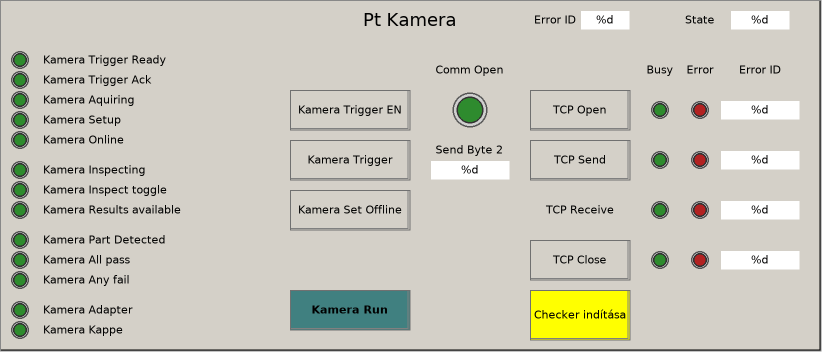
VISUALIZATION Kamera_Pt  // 822x352
    Rectangle (0,0 820x350)
    Lamp1 (450,90 40x40), variable: KAMERAREMOTE.bKameraCommOpen, style: Lamp-Lamp1-Green
    Label (530,200 100x20), "TCP Receive"
    Lamp1 (650,100 20x20), variable: KAMERAREMOTE.bConnectBusy, style: Lamp-Lamp1-Green
    Label (350,0 120x40), "Pt Kamera"
    Button (530,90 100x40), "TCP Open"
        tap KAMERAREMOTE.bKameraCommOpenEnable p1329445385=TRUE
    Button (530,240 100x40), "TCP Close"
        tap KAMERAREMOTE.bKameraCommCloseEnable
    Button (530,140 100x40), "TCP Send"
        tap KAMERAREMOTE.bKameraCommandSend
    Lamp1 (690,100 20x20), variable: KAMERAREMOTE.bConnectError, style: Lamp-Lamp1-Red
    Label (640,60 40x20), "Busy"
    Label (680,60 40x20), "Error"
    Textfield (720,100 80x20), "%d", text variable: KAMERAREMOTE.nConnectErrId
    Label (730,60 60x20), "Error ID"
    Lamp1 (650,250 20x20), variable: KAMERAREMOTE.bCloseBusy, style: Lamp-Lamp1-Green
    Lamp1 (690,250 20x20), variable: KAMERAREMOTE.bCloseError, style: Lamp-Lamp1-Red
    Textfield (720,250 80x20), "%d", text variable: KAMERAREMOTE.nCloseErrId
    Lamp1 (650,150 20x20), variable: KAMERAREMOTE.bSendBusy, style: Lamp-Lamp1-Green
    Lamp1 (690,150 20x20), variable: KAMERAREMOTE.bSendError, style: Lamp-Lamp1-Red
    Textfield (720,150 80x20), "%d", text variable: KAMERAREMOTE.nSendErrId
    Lamp1 (650,200 20x20), variable: KAMERAREMOTE.bReceiveBusy, style: Lamp-Lamp1-Green
    Lamp1 (690,200 20x20), variable: KAMERAREMOTE.bReceiveError, style: Lamp-Lamp1-Red
    Textfield (720,200 80x20), "%d", text variable: KAMERAREMOTE.nReceiveErrId
    Label (430,60 79x20), "Comm Open"
    Label (680,10 40x20), "State"
    Textfield (730,10 60x20), "%d", text variable: KAMERAREMOTE.iState
    Button (290,90 120x40), "Kamera Trigger EN"
        toggle KAMERAREMOTE.bKameraTriggerEN
    Button (290,140 120x40), "Kamera Trigger"
        toggle AUTOMATA.bKameraTrig
    Button (290,190 120x40), "Kamera Set Offline"
        toggle KAMERAREMOTE.bKameraSetOffline
    Textfield (430,160 80x20), "%d", text variable: KAMERAREMOTE.baSendByteArray[2]
    Label (430,140 79x20), "Send Byte 2"
    Label (530,10 50x20), "Error ID"
    Textfield (580,10 50x20), "%d", text variable: KameraProcess.n_OutErrId
    Lamp1 (10,50 20x20), variable: KAMERAREMOTE.bKameraTriggerReady, style: Lamp-Lamp1-Green
    Label (40,50 210x20), "Kamera Trigger Ready"
    Lamp1 (10,70 20x20), variable: KAMERAREMOTE.bKameraTriggerAck, style: Lamp-Lamp1-Green
    Label (40,70 210x20), "Kamera Trigger Ack"
    Lamp1 (10,90 20x20), variable: KAMERAREMOTE.bKameraAcquiring, style: Lamp-Lamp1-Green
    Label (40,90 210x20), "Kamera Aquiring"
    Lamp1 (10,110 20x20), variable: KAMERAREMOTE.bKameraSetup, style: Lamp-Lamp1-Green
    Label (40,110 210x20), "Kamera Setup"
    Lamp1 (10,130 20x20), variable: KAMERAREMOTE.bKameraOnline, style: Lamp-Lamp1-Green
    Label (40,130 210x20), "Kamera Online"
    Lamp1 (10,160 20x20), variable: KAMERAREMOTE.bKameraInspecting, style: Lamp-Lamp1-Green
    Label (40,160 210x20), "Kamera Inspecting"
    Lamp1 (10,180 20x20), variable: KAMERAREMOTE.bKameraInspectToggle, style: Lamp-Lamp1-Green
    Label (40,180 210x20), "Kamera Inspect toggle"
    Lamp1 (10,200 20x20), variable: KAMERAREMOTE.bKameraResultsAvble, style: Lamp-Lamp1-Green
    Label (40,200 210x20), "Kamera Results available"
    Lamp1 (10,230 20x20), variable: KAMERAREMOTE.bKameraPartDetect, style: Lamp-Lamp1-Green
    Label (40,230 210x20), "Kamera Part Detected"
    Lamp1 (10,250 20x20), variable: KAMERAREMOTE.bKameraAllPass, style: Lamp-Lamp1-Green
    Label (40,250 210x20), "Kamera All pass"
    Lamp1 (10,270 20x20), variable: KAMERAREMOTE.bKameraAnyFail, style: Lamp-Lamp1-Green
    Label (40,270 210x20), "Kamera Any fail"
    Lamp1 (10,300 20x20), variable: KAMERAREMOTE.bKameraOut04, style: Lamp-Lamp1-Green
    Label (40,300 210x20), "Kamera Adapter"
    Lamp1 (10,320 20x20), variable: KAMERAREMOTE.bKameraOut05, style: Lamp-Lamp1-Green
    Label (40,320 210x20), "Kamera Kappe"
    Button (290,290 120x40), "Kamera Run"
        toggle KameraProcess.bKameraRun
    Button (530,290 100x50), "Checker indítása", tooltip "A Pt oldali kamera saját vezérlő szoftvere", pressed state: Laser.bStartFOBADraw
        OnMouseUp: execute { KAMERAREMOTE.bStartChecker:=TRUE; }
END_VISUALIZATION

(* stored: Version 1.1.0.1, ProductVersion 3.1.4024.11
   Visu Kamera_Pt: Id {3b430e0f-bbb8-4e88-872e-7f94e07e90f2} *)
